Staubli VAL3: stopCycle.pgx

public program stopCycle()
begin
  if cycleStatus:bCycle or cycleStatus:bSimulation
    // CYCLE MOTION
    stopMove()
    logMsg("[KERNEL] CYCLE:Stop the cycle ")
    // enable the bit to stop the cycle
    cycleStatus:bToStop=true
    watch(cycleStatus:bToStop==false,1)
  endIf
end
